// Mitsubishi GX Works2 project: 240416_순시동작한시복귀   PLC: Q03UDV

PROGRAM MAIN
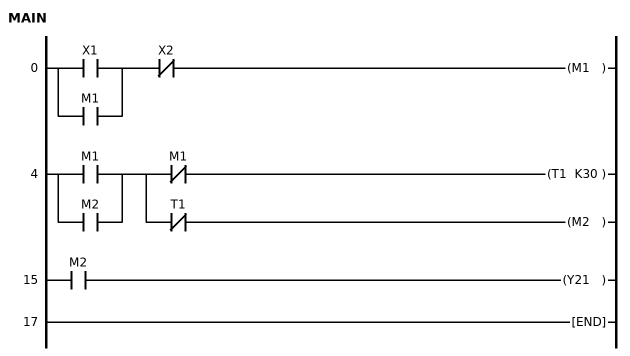
0     LD      X1
      OR      M1
      ANI     X2
      OUT     M1
4     LD      M1
      OR      M2
      MPS
      ANI     M1
      OUT     T1 K30
      MPP
      ANI     T1
      OUT     M2
15    LD      M2
      OUT     Y21
17    END
END_PROGRAM
